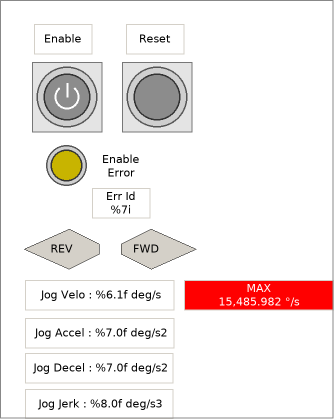
VISUALIZATION Visualization  // 334x419
    PowerSwitch (32,62 70x70), variable: MAIN.bA1Enable, behaviour: TOGGLE, style: Switch-PowerSwitch-Gray
    Lamp1 (43,142 47x47), variable: MAIN.bA1PwrErrorLatch, style: Lamp-Lamp1-Yellow
    Polygon (121,244) (151,229) (196,249) (151,269) (121,254), "FWD"
        tap MAIN.bA1JogFwd
    Polygon (99,244) (69,229) (24,249) (69,269) (99,254), "REV"
        tap MAIN.bA1JogRev
    PushSwitch (122,62 70x70), variable: MAIN.bA1Reset, behaviour: TOGGLE, style: Switch-PushSwitch-Gray
    Textfield (25,280 149x30), "Jog Velo : %6.1f deg/s", text variable: MAIN.bA1JogVelocity
        OnMouseClick: write the text variable via Default, min 0, max 15000
    Textfield (25,318 149x30), "Jog Accel : %7.0f deg/s2", text variable: MAIN.bA1JogAccel
        OnMouseClick: write the text variable via Default, min 0, max 100000
    Textfield (25,389 148x30), "Jog Jerk : %8.0f deg/s3", text variable: MAIN.bA1JogJerk
        OnMouseClick: write the text variable via Default, min 0, max 100000
    Textfield (25,353 148x30), "Jog Decel : %7.0f deg/s2", text variable: MAIN.bA1JogDecel
        OnMouseClick: write the text variable via Default, min 0, max 100000
    Textfield (126,24 58x30), "Reset"
    Textfield (34,24 58x30), "Enable"
    Textfield (92,151 58x30), "Enable Error"
    Textfield (92,188 58x30), "Err Id %7i", text variable: MAIN.bA1PwrErrorIdLatch
    Textfield (184,280 150x30), "MAX 15,485.982 °/s"
END_VISUALIZATION

(* stored: Version 1.1.0.1, ProductVersion 3.1.4026.12
   Visu Visualization: Id {0fb270fb-43af-4536-a054-13d95c2b08c6} *)
